KUKA KRL data list: FindBarrel.dat

&ACCESS RVP
&REL 1
&PARAM DISKPATH = KRC:\R1\Program\Production\Utilities
DEFDAT  FindBarrel
;FOLD EXTERNAL DECLARATIONS;%{PE}%MKUKATPBASIS,%CEXT,%VCOMMON,%P
;FOLD BASISTECH EXT;%{PE}%MKUKATPBASIS,%CEXT,%VEXT,%P
EXT  BAS (BAS_COMMAND  :IN,REAL  :IN )
;ENDFOLD (BASISTECH EXT)
;FOLD USER EXT;%{E}%MKUKATPUSER,%CEXT,%VEXT,%P
;Make your modifications here
;ENDFOLD (USER EXT)
;ENDFOLD (EXTERNAL DECLARATIONS)
DECL INT COUNTER=4
DECL INT MINCOUNT=2
DECL INT MAXCOUNT=12

ENDDAT
